// TIA Portal V20 export
DATA_BLOCK "DB_Temperature"   // DB490
// stored: AutoNumber false, InstanceOfName FB_Temperature, InstanceOfType FB
"FB_Temperature"
   // VAR
   //    sPIDRestart : Bool;
   //    sPIDHoldI : Bool;
   //    sXAxisWarning : Real;
   //    sPIDClimOut : Real;
   //    sP : Real;
   //    sI : Time;
   //    sD : Time;
   //    sTimeOutFlowChiller : TON_TIME;
   //    sTimeOutLevelChiller { S7_SetPoint := 'True'} : TON_TIME;
   //    sTimeOutChillerGood : TON_TIME;
   //    sTimeOutCooling : TON_TIME;
   //    sTemperature_X_PT1000 { S7_SetPoint := 'True'} : "FB_AnalogInputThreshold";
   //    sTemperature_Y_PT1000 { S7_SetPoint := 'True'} : "FB_AnalogInputThreshold";
   //    sAmbiantTemperature { S7_SetPoint := 'True'} : "FB_AnalogInputThreshold";
   //    sMachineTemperature { S7_SetPoint := 'True'} : "FB_AnalogInputThreshold";
   //    sCabinetTemperatureMeasure { S7_SetPoint := 'True'} : "FB_AnalogInputThreshold";
   //    sColdWaterTemperatureInput { S7_SetPoint := 'True'} : "FB_AnalogInputThreshold";
   //    sColdWaterTemperatureOutput { S7_SetPoint := 'True'} : "FB_AnalogInputThreshold";
   //    sTemperatureCooling { S7_SetPoint := 'True'} : "FB_AnalogInputThreshold";
   // END_VAR
BEGIN
END_DATA_BLOCK
